{attribute addProperty BoxType "ELM3002-0000-0016"}
{attribute addProperty Id "LowUDINT3241HiUDINT3242"}
{attribute addProperty CRC "896265644"}
{attribute addProperty SizeInBites "64"}
{attribute addProperty SizeInBytes "8"}
TYPE StartTimeNextLatch_356BEDAC :
STRUCT
	{attribute addProperty Name "Low"}
	Low : UDINT;
	{attribute addProperty Name "Hi"}
	Hi : UDINT;
END_STRUCT
END_TYPE

(* stored: Version 1.2.0.0, ProductVersion 3.1.4024.9
   DUT StartTimeNextLatch_356BEDAC: Id {76647d3b-7bce-4365-bf86-59ea97b9789a} *)
